PROGRAM pouMcAlarms
VAR
	idbMsgAlarm: FB_CheckMessageBounds;

END_VAR

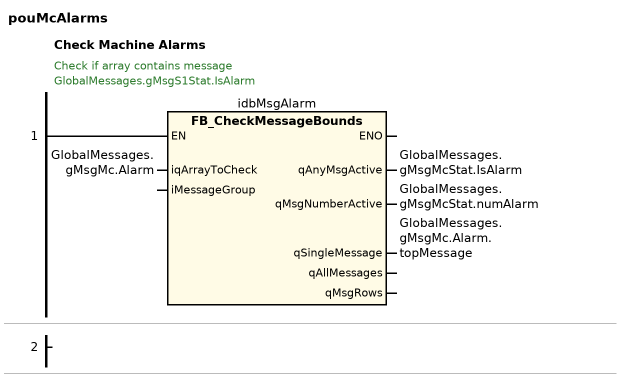
// NETWORK 1: Check Machine Alarms
// Check if array contains message
//
// GlobalMessages.gMsgS1Stat.IsAlarm
idbMsgAlarm(
    iqArrayToCheck := GlobalMessages.gMsgMc.Alarm,
    qAnyMsgActive => GlobalMessages.gMsgMcStat.IsAlarm,
    qMsgNumberActive => GlobalMessages.gMsgMcStat.numAlarm,
    qSingleMessage => GlobalMessages.gMsgMc.Alarm.topMessage); // FB_CheckMessageBounds

// NETWORK 2

END_PROGRAM

(* stored: Version 1.1.0.1, ProductVersion 3.1.4024.12
   POU pouMcAlarms: Id {3f0fd1a1-2fbb-4f59-9ec9-208cf01105f8}, SpecialFunc None *)
